# B&R Automation Studio project Lab2
Automation Studio 

## Logical view

### Library Logical/DriveLib (ANSIC)

#### Types.typ - Exported data types
```iecst
TYPE
	EN_DoorStates :
		(
		ST_INIT := 0,
		ST_UNKNOWN := 1,
		ST_OPEN := 2,
		ST_CLOSE := 6,
		ST_ACC_POS := 3,
		ST_ACC_NEG := 7,
		ST_POS := 4,
		ST_NEG := 8,
		ST_DEC_POS := 5,
		ST_DEC_NEG := 9
		);
	driveComands :
		(
		CMD_SWITCHED_ON := 7,
		CMD_DISABLE_VOLTAGE := 0,
		CMD_ENABLED := 15,
		CMD_SHUTDOWN := 6,
		STATE_READY := 33,
		STATE_DISABLED := 64,
		STATE_SWITCHED_ON := 35
		);
END_TYPE
```

#### DriveLib.fun - Exported functions and function blocks
```iecst
{REDUND_ERROR} {REDUND_UNREPLICABLE} FUNCTION_BLOCK FB_DriveStateMashine (*TODO: Add your comment here*) (*$GROUP=User,$CAT=User,$GROUPICON=User.png,$CATICON=User.png*)
	VAR_INPUT
		state : {REDUND_UNREPLICABLE} UINT; (*Sostiyanie chastotnogo preobrazovatelya*)
		enable : {REDUND_UNREPLICABLE} BOOL; (*Signal raboti FunchBlock*)
	END_VAR
	VAR_OUTPUT
		command : {REDUND_UNREPLICABLE} UINT; (*Comand, podavayemaya na chastotniy preobrazovatel*)
		speed : {REDUND_UNREPLICABLE} INT; (*Zadannaya skorosti*)
	END_VAR
END_FUNCTION_BLOCK

{REDUND_ERROR} FUNCTION_BLOCK FB_DoorStateMashine (*TODO: Add your comment here*) (*$GROUP=User,$CAT=User,$GROUPICON=User.png,$CATICON=User.png*)
	VAR_INPUT
		state : {REDUND_UNREPLICABLE} UINT; (*sostoyanie chastotnogo preobrazovatelya*)
		sw1 : {REDUND_UNREPLICABLE} BOOL; (*Signal konc switch1*)
		sw2 : {REDUND_UNREPLICABLE} BOOL; (*Signal konc switch2*)
		sw3 : {REDUND_UNREPLICABLE} BOOL; (*Signal konc switch3*)
		sw4 : {REDUND_UNREPLICABLE} BOOL; (*Signal konc switch4*)
		direction : {REDUND_UNREPLICABLE} BOOL; (*comand, podavayemaya na chast preobr*)
	END_VAR
	VAR
		swo1 : BOOL; (*Old Signal konc switch1*)
		swo2 : BOOL; (*Old Signal konc switch2*)
		swo3 : BOOL; (*Old Signal konc switch3*)
		swo4 : BOOL; (*Old Signal konc switch4*)
	END_VAR
	VAR_OUTPUT
		speed : {REDUND_UNREPLICABLE} INT; (*zadannaya skorosty*)
	END_VAR
END_FUNCTION_BLOCK

{REDUND_ERROR} {REDUND_UNREPLICABLE} FUNCTION_BLOCK FB_LedStateMashine (*TODO: Add your comment here*) (*$GROUP=User,$CAT=User,$GROUPICON=User.png,$CATICON=User.png*)
	VAR_INPUT
		state : {REDUND_UNREPLICABLE} UINT; (*sostoyaniye chast preobr*)
	END_VAR
	VAR_OUTPUT
		led1 : {REDUND_UNREPLICABLE} BOOL; (*Signal raboti FB*)
		led2 : {REDUND_UNREPLICABLE} BOOL; (*Signal raboti FB*)
		led3 : {REDUND_UNREPLICABLE} BOOL; (*Signal raboti FB*)
		led4 : {REDUND_UNREPLICABLE} BOOL; (*Signal raboti FB*)
		timer : {REDUND_UNREPLICABLE} INT; (*Zadannaya skorosty*)
	END_VAR
END_FUNCTION_BLOCK
```

#### FB_DriveStateMashine.c
```c
#include <bur/plctypes.h>
#ifdef __cplusplus
	extern "C"
	{
#endif
	#include "DriveLib.h"
#ifdef __cplusplus
	};
#endif
/* TODO: Add your comment here */
void FB_DriveStateMashine(struct FB_DriveStateMashine* inst)
{
	/*TODO: Add your code here*/
	UINT mask = inst->state & 0x6f;
	if(!inst->enable)
	{
		inst->command = CMD_SHUTDOWN;
	}
	else
	{
		switch (mask)
		{
			case STATE_DISABLED:
				inst->command = CMD_SHUTDOWN;
				break;

			case STATE_READY:
				inst->command = CMD_ENABLED;
				break;

			case STATE_SWITCHED_ON:
				inst->command = CMD_SWITCHED_ON;
				break;
		}
	}
}
```

#### FB_DoorStateMashine.c
```c
#include <bur/plctypes.h>
#ifdef __cplusplus
	extern "C"
	{
#endif
	#include "DriveLib.h"
#ifdef __cplusplus
	};
#endif
/* TODO: Add your comment here */
void FB_DoorStateMashine(struct FB_DoorStateMashine* inst)
{
	/*TODO: Add your code here*/
	switch(inst->state)
	{
		case ST_INIT:
			{
				if(inst->sw1==0 && inst->sw2==0 && inst->sw3==0 && inst->sw4==0)
					inst->state=ST_UNKNOWN;
				break;
			}
		case ST_UNKNOWN:
			{
				if(inst->direction==0 && inst->sw1!=inst->swo1)
					inst->state=ST_CLOSE;
				if(inst->direction==1 && inst->sw1!=inst->swo1)
					inst->state=ST_NEG;
				if(inst->direction==1 && inst->sw2!=inst->swo2)
					inst->state=ST_ACC_NEG;
				if(inst->direction==1 && inst->sw3!=inst->swo3)
					inst->state=ST_DEC_NEG;

				if(inst->direction==1 && inst->sw4!=inst->swo4)
					inst->state=ST_OPEN;
				if(inst->direction==0 && inst->sw4!=inst->swo4)
					inst->state=ST_POS;
				if(inst->direction==0 && inst->sw3!=inst->swo3)
					inst->state=ST_ACC_POS;
				if(inst->direction==0 && inst->sw2!=inst->swo2)
					inst->state=ST_DEC_POS;
				break;
			}

		case ST_CLOSE:
			{
				inst->speed = 0;
				if(inst->direction==1)
					inst->state=ST_NEG;
				break;
			}
		case ST_NEG:
			{
				inst->speed = -200;
				if(inst->direction==1 && inst->sw2!=inst->swo2)
					inst->state=ST_ACC_NEG;
				if(inst->direction==0)
					inst->state=ST_DEC_POS;
				break;

			}
		case ST_ACC_NEG:
			{
				inst->speed = -600;
				if(inst->direction==1 && inst->sw3!=inst->swo3)
					inst->state=ST_DEC_NEG;
				if(inst->direction==0)
					inst->state=ST_ACC_POS;
				break;
			}
		case ST_DEC_NEG:
			{
				inst->speed = -200;
				if(inst->direction==1 && inst->sw4!=inst->swo4)
					inst->state=ST_OPEN;
				if(inst->direction==0)
					inst->state=ST_POS;
				break;
			}

		case ST_OPEN:
			{
				inst->speed = 0;
				if(inst->direction==0)
					inst->state=ST_POS;
				break;
			}
		case ST_POS:
			{
				inst->speed = 200;
				if(inst->direction==0 && inst->sw3!=inst->swo3)
					inst->state=ST_ACC_POS;
				if(inst->direction==1)
					inst->state=ST_DEC_NEG;
				break;
			}
		case ST_ACC_POS:
			{
				inst->speed = 600;
				if(inst->direction==0 && inst->sw2!=inst->swo2)
					inst->state=ST_DEC_POS;
				if(inst->direction==1)
					inst->state=ST_ACC_NEG;
				break;
			}
		case ST_DEC_POS:
			{
				inst->speed = 200;
				if(inst->direction==0 && inst->sw1!=inst->swo1)
					inst->state=ST_CLOSE;
				if(inst->direction==1)
					inst->state=ST_NEG;

				break;
			}
	}

	inst->swo1=inst->sw1;
	inst->swo2=inst->sw2;
	inst->swo3=inst->sw3;
	inst->swo4=inst->sw4;
}
```

#### FB_LedStateMashine.c
```c
#include <bur/plctypes.h>
#ifdef __cplusplus
	extern "C"
	{
#endif
	#include "DriveLib.h"
#ifdef __cplusplus
	};
#endif
/* TODO: Add your comment here */
void FB_LedStateMashine(struct FB_LedStateMashine* inst)
{
	/*TODO: Add your code here*/
	switch(inst->state)
	{
		case ST_INIT:
			{

				break;
			}

		case ST_UNKNOWN:
			{
				if(inst->timer%5==4)
				{
					inst->led1=!inst->led1;
					inst->led2=!inst->led2;
					inst->led3=!inst->led3;
					inst->led4=!inst->led4;
				}
				break;
			}

		case ST_CLOSE:
			{
				inst->led1=1;
				inst->led2=1;
				inst->led3=1;
				inst->led4=1;
				break;
			}
		case ST_NEG:
			{
				inst->led1=0;
				if(inst->timer%10==9)
					inst->led2=!inst->led2;
				inst->led3=1;
				inst->led4=1;
				break;
			}
		case ST_ACC_NEG:
			{
				inst->led1=0;
				inst->led2=0;
				if(inst->timer%5==4)
					inst->led3=!inst->led3;
				inst->led4=1;
				break;
			}
		case ST_DEC_NEG:
			{
				inst->led1=0;
				inst->led2=0;
				inst->led3=0;
				if(inst->timer%10==9)
					inst->led4=!inst->led4;
				break;
			}

		case ST_OPEN:
			{
				inst->led1=0;
				inst->led2=0;
				inst->led3=0;
				inst->led4=0;
				break;
			}
		case ST_POS:
			{
				inst->led1=0;
				inst->led2=0;
				if(inst->timer%10==9)
					inst->led3=!inst->led3;
				inst->led4=1;
				break;
			}
		case ST_ACC_POS:
			{
				inst->led1=0;
				if(inst->timer%5==4)
					inst->led2=!inst->led2;
				inst->led3=1;
				inst->led4=1;
				break;
			}
		case ST_DEC_POS:
			{
				if(inst->timer%10==9)
					inst->led1=!inst->led1;
				inst->led2=1;
				inst->led3=1;
				inst->led4=1;
				break;
			}
	}
	inst->timer++;
}
```

### Program Logical/Program

#### Variables.var
```iecst
VAR
	stateMachine : EN_DoorStates := ST_INIT;
	doorSM : FB_DoorStateMashine := (0);
	motorSM : FB_DriveStateMashine := (0);
	ledSM : FB_LedStateMashine := (0);
END_VAR
```

#### Cyclic.c
```c
#include <bur/plctypes.h>

#ifdef _DEFAULT_INCLUDES
	#include <AsDefault.h>
#endif

void _CYCLIC ProgramCyclic(void)
{
	FB_DoorStateMashine(&doorSM);
	motorSM.speed = doorSM.speed;
	FB_DriveStateMashine(&motorSM);
	ledSM.state = doorSM.state;
	FB_LedStateMashine(&ledSM);
}
```

#### Init.c
```c
#include <bur/plctypes.h>

#ifdef _DEFAULT_INCLUDES
	#include <AsDefault.h>
#endif

void _INIT ProgramInit(void)
{
	motorSM.enable=1;
}
```

Listed in the project but not available here: Logical/DriveLib/Constants.var
